FUNCTION_BLOCK counter2 (* Basic Function Block Type *)
  (* Standard: 61499-2 *)
  (* Version 0.0, 5/24/2016, gulzha, nxtControl GmbH, Template *)
  PACKAGE Main;
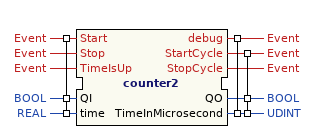
  EVENT_INPUT
    Start WITH QI, time;
    Stop;
    TimeIsUp;
  END_EVENT
  EVENT_OUTPUT
    debug WITH TimeInMicrosecond;
    StartCycle WITH QO, TimeInMicrosecond;
    StopCycle;
  END_EVENT
  VAR_INPUT
    QI : BOOL; (* Input event qualifier *)
    time : REAL; (* in seconds *)
  END_VAR
  VAR_OUTPUT
    QO : BOOL; (* Output event qualifier *)
    TimeInMicrosecond : UDINT;
  END_VAR
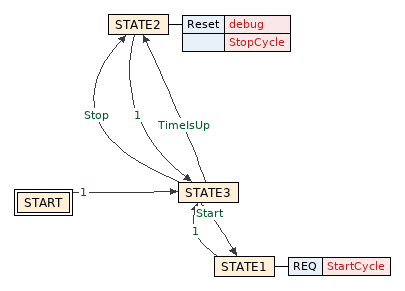
  EC_STATES
    START; (* Initial State *)
    STATE2 : Reset -> debug, -> StopCycle;
    STATE3;
    STATE1 : REQ -> StartCycle;
  END_STATES
  EC_TRANSITIONS
    START TO STATE3 := 1;
    STATE3 TO STATE2 := Stop;
    STATE3 TO STATE2 := TimeIsUp;
    STATE3 TO STATE1 := Start;
    STATE1 TO STATE3 := 1;
    STATE2 TO STATE3 := 1;
  END_TRANSITIONS
  ALGORITHM REQ IN ST: (* Normally executed algorithm *)
;


TimeInMicrosecond := REAL_TO_UDINT(time*1000000);
TimeInMicrosecond := TimeInMicrosecond/2;
  END_ALGORITHM
  ALGORITHM Reset IN ST:
;

TimeInMicrosecond := 0;
  END_ALGORITHM
END_FUNCTION_BLOCK
